TYPE ST_ScrewdriverProcessConfig :
STRUCT
    tPreTightenSimulation : TIME;
    tFinalTightenSimulation : TIME;
END_STRUCT
END_TYPE

(* stored: Version 1.1.0.1, ProductVersion 3.1.4026.20
   DUT ST_ScrewdriverProcessConfig: Id {1232b83f-db07-4368-ba3a-b14a8f7af5f2} *)
